INTERFACE I_EcSlaveInfoData EXTENDS __SYSTEM.IQueryInterface

PROPERTY PUBLIC rInfoData : reference to EcSlaveInfoData
GET
END_GET
END_PROPERTY

END_INTERFACE

(* stored: Version 1.1.0.1, ProductVersion 3.1.4024.4
   Itf I_EcSlaveInfoData: Id {5706b104-2ae8-4159-b5a9-4cb9cf0427b9}
   Property rInfoData: Id {a4e23c19-ff21-443d-990c-1a7c92151b0d}
   Get Get: Id {c083f74d-f681-4919-bf91-4ecbf91112f6} *)
